	        #sFB_MCOConveyLinxAixController_110(iUDT_AixConfig          := #iqUDT_Configuration."110".MCO_M01,
	                                            iv_AixInputsModule    := #iUDT_MotorInput110,
	                                            ix_24vOk                := #ix_24vOk,
	                                            ix_SimulationModeActive := "DB_Memory".Simulation,
	                                            ii_MotorPositionId      := 1,
	                                            qUDT_HMIStatus          => #iqUDT_WorkstationStatus."110".MCO_M01,
	                                            iqv_AixOutputsModule  := #iqUDT_MotorOutput110,
	                                            iqUDT_ConveyorInterface := #sUDT_Interface_110,
	                                            iqUDT_MCOStatistics     := #iqUDT_WorkstationStatistics."110".MCO_M01);
	    END_REGION

	END_REGION

	REGION 120

	    REGION Displacement
	        #sFB_Displacement120(#sUDT_Interface_120);
	    END_REGION

	    REGION Tracking

	        #sFB_Tracking_120(iUDT_ConveyorCommonConfiguration := #iqUDT_Configuration."120".Conveyor.Common,
	                          iqa_TrackingData                 := #sa_TrackingArray_120,
	                          iqUDT_ConveyorInterface          := #sUDT_Interface_120,
	                          iqUDT_HandshakeUp                := #sUDT_Handshake_110,
	                          iqUDT_Handshake                  := #sUDT_Handshake_120);

	    END_REGION

	    REGION EoS

	        #sFB_PECUpdate_120(iUDT_PECUpdateConfiguration      := #iqUDT_Configuration."120".PEC_EoS,
	                           iUDT_ConveyorCommonConfiguration := #iqUDT_Configuration."120".Conveyor.Common,
	                           ix_PEC                           := #iUDT_MotorInput110.AllSensorPortInputs.RightSensor,
	                           ix_TeachingMode                  := FALSE,
	                           qUDT_Status                      => #iqUDT_WorkstationStatus."120".PEC_EoS,
	                           iqUDT_ConveyorInterface          := #sUDT_Interface_120,
	                           iqUDT_UnknownGINRange            := #iqUDT_UnknownGINRange,
	                           iqUDT_FifoHeader                 := #sUDT_FifoLostGINHeader,
	                           iqUDT_Statistics                 := #iqUDT_WorkstationStatistics."120".PEC_EoS,
	                           iqa_TrackingData                 := #sa_TrackingArray_120,
	                           iqa_FifoData                     := #sa_FifoLostGINData);

	    END_REGION

	    REGION Conveyor

	        #sFB_Conveyor_120(iUDT_ConveyorConfiguration := #iqUDT_Configuration."120".Conveyor,
	                          idi_PECEoSDistance         := #iqUDT_Configuration."120".PEC_EoS.Distance,
	                          idi_PECBoSDistance         := 0,
	                          ii_ExternalSpeed           := 0,
	                          ix_SafetyOk                := #ix_SafetyOk,
	                          ix_24vOk                   := #ix_24vOk,
	                          ix_400vOk                  := #ix_400vOk,
	                          ix_HardwareOk              := #iUDT_HardwareOk."110",
	                          ix_PECEoS                  := #iqUDT_WorkstationStatus."120".PEC_EoS.PEC,
	                          ix_PECBoS                  := TRUE,
	                          ix_ReverseDirection        := FALSE,
	                          ix_ExternalRequestDieBack  := #sx_Hold120 OR (#sUDT_Interface_130.ActualSpeed = 0 AND NOT #iqUDT_WorkstationStatus."120".PEC_EoS.PEC),
	                          ix_ExternalRequestHold     := FALSE,
	                          ix_ResetEnergySave         := FALSE,
	                          qUDT_HMIStatus             => #iqUDT_WorkstationStatus."120".Conveyor,
	                          qUDT_Status                => #iqUDT_WorkstationCommonStatus."120",
	                          iqUDT_EquipmentControl     := #iqUDT_EquipmentControl,
	                          iqUDT_ConveyorCommand      := #iqUDT_WorkstationCommands."120".Conveyor,
	                          iqUDT_ConveyorInterface    := #sUDT_Interface_120,
	                          iqUDT_HandShakeUp          := #sUDT_Handshake_110,
	                          iqUDT_HandShake            := #sUDT_Handshake_120,
	                          iqUDT_Statistics           := #iqUDT_WorkstationStatistics."120".Conveyor);

	    END_REGION

	    REGION MCO

	        #sFB_MCOConveyLinxAixController_120(iUDT_AixConfig          := #iqUDT_Configuration."120".MCO_M01,
	                                            iv_AixInputsModule    := #iUDT_MotorInput110,
	                                            ix_24vOk                := #ix_24vOk,
	                                            ix_SimulationModeActive := "DB_Memory".Simulation,
	                                            ii_MotorPositionId      := 2,
	                                            qUDT_HMIStatus          => #iqUDT_WorkstationStatus."120".MCO_M01,
	                                            iqv_AixOutputsModule  := #iqUDT_MotorOutput110,
	                                            iqUDT_ConveyorInterface := #sUDT_Interface_120,
	                                            iqUDT_MCOStatistics     := #iqUDT_WorkstationStatistics."120".MCO_M01);
	    END_REGION

	END_REGION

	REGION 130

	    REGION Displacement
	        #sFB_Displacement130(#sUDT_Interface_130);
	    END_REGION

	    REGION Tracking

	        #sFB_Tracking_130(iUDT_ConveyorCommonConfiguration := #iqUDT_Configuration."130".Conveyor.Common,
	                          iqa_TrackingData                 := #sa_TrackingArray_130,
	                          iqUDT_ConveyorInterface          := #sUDT_Interface_130,
	                          iqUDT_HandshakeUp                := #sUDT_Handshake_120,
	                          iqUDT_Handshake                  := #sUDT_Handshake_130);

	    END_REGION

	    REGION EoS

	        #sFB_PECUpdate_130(iUDT_PECUpdateConfiguration      := #iqUDT_Configuration."130".PEC_EoS,
	                           iUDT_ConveyorCommonConfiguration := #iqUDT_Configuration."130".Conveyor.Common,
	                           ix_PEC                           := #iUDT_MotorInput130.AllSensorPortInputs.LeftSensor,
	                           ix_TeachingMode                  := FALSE,
	                           qUDT_Status                      => #iqUDT_WorkstationStatus."130".PEC_EoS,
	                           iqUDT_ConveyorInterface          := #sUDT_Interface_130,
	                           iqUDT_UnknownGINRange            := #iqUDT_UnknownGINRange,
	                           iqUDT_FifoHeader                 := #sUDT_FifoLostGINHeader,
	                           iqUDT_Statistics                 := #iqUDT_WorkstationStatistics."130".PEC_EoS,
	                           iqa_TrackingData                 := #sa_TrackingArray_130,
	                           iqa_FifoData                     := #sa_FifoLostGINData);

	    END_REGION

	    REGION Conveyor

	        #sUDT_Handshake_130.RTR := #sUDT_Handshake_130.RTR AND NOT #sx_Hold130 OR #iqUDT_WorkstationStatus."130".PEC_EoS.PEC;

	        #sFB_Conveyor_130(iUDT_ConveyorConfiguration := #iqUDT_Configuration."130".Conveyor,
	                          idi_PECEoSDistance         := #iqUDT_Configuration."130".PEC_EoS.Distance,
	                          idi_PECBoSDistance         := 0,
	                          ii_ExternalSpeed           := 0,
	                          ix_SafetyOk                := #ix_SafetyOk,
	                          ix_24vOk                   := #ix_24vOk,
	                          ix_400vOk                  := #ix_400vOk,
	                          ix_HardwareOk              := #iUDT_HardwareOk."130",
	                          ix_PECEoS                  := #iqUDT_WorkstationStatus."130".PEC_EoS.PEC,
	                          ix_PECBoS                  := TRUE,
	                          ix_ReverseDirection        := FALSE,
	                          ix_ExternalRequestDieBack  := FALSE,
	                          ix_ExternalRequestHold     := #sx_Hold130,
	                          ix_ResetEnergySave         := FALSE,
	                          qUDT_HMIStatus             => #iqUDT_WorkstationStatus."130".Conveyor,
	                          qUDT_Status                => #iqUDT_WorkstationCommonStatus."130",
	                          iqUDT_EquipmentControl     := #iqUDT_EquipmentControl,
	                          iqUDT_ConveyorCommand      := #iqUDT_WorkstationCommands."130".Conveyor,
	                          iqUDT_ConveyorInterface    := #sUDT_Interface_130,
	                          iqUDT_HandShakeUp          := #sUDT_Handshake_120,
	                          iqUDT_HandShake            := #sUDT_Handshake_130,
	                          iqUDT_Statistics           := #iqUDT_WorkstationStatistics."130".Conveyor);


	    END_REGION

	    REGION MCO

	        #sFB_MCOConveyLinxAixController_130(iUDT_AixConfig          := #iqUDT_Configuration."130".MCO_M01,
	                                            iv_AixInputsModule    := #iUDT_MotorInput130,
	                                            ix_24vOk                := #ix_24vOk,
	                                            ix_SimulationModeActive := "DB_Memory".Simulation,
	                                            ii_MotorPositionId      := 1,
	                                            qUDT_HMIStatus          => #iqUDT_WorkstationStatus."130".MCO_M01,
	                                            iqv_AixOutputsModule  := #iqUDT_MotorOutput130,
	                                            iqUDT_ConveyorInterface := #sUDT_Interface_130,
	                                            iqUDT_MCOStatistics     := #iqUDT_WorkstationStatistics."130".MCO_M01);
	    END_REGION

	END_REGION

	REGION 140

	    REGION Displacement
	        #sFB_Displacement140(#sUDT_Interface_140);
	    END_REGION

	    REGION MCO

	        #sFB_MCOConveyLinxAixController_140(iUDT_AixConfig          := #iqUDT_Configuration."140".MCO_M01,
	                                            iv_AixInputsModule    := #iUDT_MotorInput140,
	                                            ii_PositionSetpoint     := #iqUDT_RATPositioning140.Lower.EndPosition,
	                                            ix_24vOk                := #ix_24vOk,
	                                            ix_SimulationModeActive := "DB_Memory".Simulation,
	                                            ii_MotorPositionId      := 1,
	                                            ix_StartPositioning     := #iqUDT_RATPositioning140.Lower.Start,
	                                            ix_ResetPosition        := #iqUDT_RATPositioning140.Lower.ResetPosition,
	                                            qUDT_HMIStatus          => #iqUDT_WorkstationStatus."140".MCO_M01,
	                                            qx_Positioned           => #iqUDT_RATPositioning140.Lower.Done,
	                                            iqv_AixOutputsModule  := #iqUDT_MotorOutput140,
	                                            iqUDT_ConveyorInterface := #sUDT_Interface_140,
	                                            iqUDT_MCOStatistics     := #iqUDT_WorkstationStatistics."140".MCO_M01);
	    END_REGION

	    REGION BladeStopEoS

	        IF (#iqUDT_Configuration.GlobalConfig.StationVariant = 2 OR #iqUDT_Configuration.GlobalConfig.StationVariant = 4 OR #iqUDT_Configuration.GlobalConfig.StationVariant = 6) THEN

	            #sFB_BladeStopEoS_140(iUDT_Configuration     := #iqUDT_Configuration."140".BladeStopEoS,
	                                  ix_IsOpened            := #ix_BladeStopIsUp140,
	                                  ix_IsClosed            := #ix_BladeStopIsDown140,
	                                  ix_AirPressureOk       := TRUE,
	                                  qx_Open                => #qx_BladeStopControl140,
	                                  qUDT_HMIStatus         => #iqUDT_WorkstationStatus."140".BladeStopEoS,
	                                  iqUDT_Statistics       := #iqUDT_WorkstationStatistics."140".BladeStopEoS,
	                                  iqUDT_EquipmentControl := #iqUDT_EquipmentControl,
	                                  iqUDT_HMICommand       := #iqUDT_WorkstationCommands."140".BladeStopEoS,
	                                  iqUDT_Interface        := #sUDT_Interface_140_BladeStopEoS);
	        END_IF;

	    END_REGION

	END_REGION

	REGION 141

	    REGION Displacement
	        #sFB_Displacement141(#sUDT_Interface_141);
	    END_REGION

	    REGION RAT

	        // #iqUDT_Configuration."141".RightAngledTransfer.BladeStop := #iqUDT_Configuration.GlobalConfig.StationVariant = 1
	        // OR #iqUDT_Configuration.GlobalConfig.StationVariant = 2
	        // OR #iqUDT_Configuration.GlobalConfig.StationVariant = 3
	        // OR #iqUDT_Configuration.GlobalConfig.StationVariant = 4;


	        IF #iqUDT_Configuration.GlobalConfig.StationVariant = 1 OR #iqUDT_Configuration.GlobalConfig.StationVariant = 3 OR #iqUDT_Configuration.GlobalConfig.StationVariant = 5 THEN
	            #sUDT_Handshake_141D := #sUDT_Handshake_241D;
	        ELSIF #iqUDT_Configuration.GlobalConfig.StationVariant = 2 OR #iqUDT_Configuration.GlobalConfig.StationVariant = 4 OR #iqUDT_Configuration.GlobalConfig.StationVariant = 6 THEN
	            #sUDT_Handshake_141C := #sUDT_Handshake_241C;
	        END_IF;

	        #sFB_RightAngledTransfer_141(iUDT_Configuration              := #iqUDT_Configuration."141".RightAngledTransfer,
	                                     iUDT_LowerConveyorConfiguration := #iqUDT_Configuration."140".Conveyor,
	                                     iUDT_UpperConveyorConfiguration := #iqUDT_Configuration."141".Conveyor,
	                                     iUDT_PECConfiguration           := #iqUDT_Configuration."140".PEC_EoS,
	                                     ii_DestinationA                 := #si_140DestinationA,
	                                     ii_DestinationB                 := #si_140DestinationB,
	                                     ii_DestinationC                 := #si_140DestinationC,
	                                     ii_DestinationD                 := #si_140DestinationD,
	                                     ix_HardwareOk                   := #iUDT_HardwareOk."140",
	                                     ix_400vOk                       := #ix_400vOk,
	                                     ix_24vOk                        := #ix_24vOk,
	                                     ix_SafetyOk                     := #ix_SafetyOk,
	                                     ix_AirPressureOk                := #ix_AirPressureOk,
	                                     ix_SectionIsDown                := #ix_SectionIsDown141,
	                                     ix_SectionIsUp                  := #ix_SectionIsUp141,
	                                     ix_ConveyorAAuto                := #iqUDT_WorkstationCommonStatus."130".AutoON,
	                                     ix_ConveyorBAuto                := #iqUDT_WorkstationCommonStatus."150".AutoON,
	                                     ix_ConveyorCAuto                := #iqUDT_WorkstationCommonStatus."241".AutoON AND (#iqUDT_Configuration.GlobalConfig.StationVariant = 2 OR #iqUDT_Configuration.GlobalConfig.StationVariant = 4 OR #iqUDT_Configuration.GlobalConfig.StationVariant = 6),
	                                     ix_ConveyorDAuto                := #iqUDT_WorkstationCommonStatus."241".AutoON AND (#iqUDT_Configuration.GlobalConfig.StationVariant = 1 OR #iqUDT_Configuration.GlobalConfig.StationVariant = 3 OR #iqUDT_Configuration.GlobalConfig.StationVariant = 5),
	                                     ix_PEC                          := #iUDT_MotorInput140.AllSensorPortInputs.LeftSensor,
	                                     ix_ExternalReceiveRequestA      := NOT #iqUDT_WorkstationStatus."130".PEC_EoS.PEC AND #sx_Enable1X0In,
	                                     ix_ExternalReceiveRequestB      := false,
	                                     ix_ExternalReceiveRequestC      := #sFB_RightAngledTransfer_241.qx_ExternalSendRequestC AND (#iqUDT_Configuration.GlobalConfig.StationVariant = 2 OR #iqUDT_Configuration.GlobalConfig.StationVariant = 4 OR #iqUDT_Configuration.GlobalConfig.StationVariant = 6),
	                                     ix_ExternalReceiveRequestD      := #sFB_RightAngledTransfer_241.qx_ExternalSendRequestD AND (#iqUDT_Configuration.GlobalConfig.StationVariant = 1 OR #iqUDT_Configuration.GlobalConfig.StationVariant = 3 OR #iqUDT_Configuration.GlobalConfig.StationVariant = 5),
	                                     ix_PECInfeedA                   := #iqUDT_WorkstationStatus."130".PEC_EoS.PEC,
	                                     ix_PECInfeedC                   := #iqUDT_WorkstationStatus."240".PEC_EoS.PEC AND (#iqUDT_Configuration.GlobalConfig.StationVariant = 2 OR #iqUDT_Configuration.GlobalConfig.StationVariant = 4 OR #iqUDT_Configuration.GlobalConfig.StationVariant = 6),
	                                     ix_PECInfeedD                   := #iqUDT_WorkstationStatus."240".PEC_EoS.PEC AND (#iqUDT_Configuration.GlobalConfig.StationVariant = 1 OR #iqUDT_Configuration.GlobalConfig.StationVariant = 3 OR #iqUDT_Configuration.GlobalConfig.StationVariant = 5),
	                                     qUDT_HMIRATStatus               => #iqUDT_WorkstationStatus."141".RightAngledTransfer,
	                                     qUDT_HMIConveyorStatus          => #iqUDT_WorkstationStatus."140".Conveyor,
	                                     qUDT_HMIPECStatus               => #iqUDT_WorkstationStatus."140".PEC_EoS,
	                                     qUDT_RATStatus                  => #iqUDT_WorkstationCommonStatus."141",
	                                     qUDT_ConveyorStatus             => #iqUDT_WorkstationCommonStatus."140",
	                                     qx_PopupControl                 => #qx_PopupControl141,
	                                     iqUDT_EquipmentControl          := #iqUDT_EquipmentControl,
	                                     iqUDT_RATCommand                := #iqUDT_WorkstationCommands."141".RightAngledTransfer,
	                                     iqUDT_ConveyorCommand           := #iqUDT_WorkstationCommands."140".Conveyor,
	                                     iqUDT_RATStatistics             := #iqUDT_WorkstationStatistics."141".RightAngledTransfer,
	                                     iqUDT_ConveyorStatistics        := #iqUDT_WorkstationStatistics."140".Conveyor,
	                                     iqUDT_PECStatistics             := #iqUDT_WorkstationStatistics."140".PEC_EoS,
	                                     iqUDT_HandShakeConveyorA        := #sUDT_Handshake_130,
	                                     iqUDT_HandShakeConveyorB        := #sUDT_Handshake_140,
	                                     iqUDT_HandShakeConveyorC        := #sUDT_Handshake_141C,
	                                     iqUDT_HandShakeConveyorD        := #sUDT_Handshake_141D,
	                                     iqUDT_LowerConveyorInterface    := #sUDT_Interface_140,
	                                     iqUDT_UpperConveyorInterface    := #sUDT_Interface_141,
	                                     iqUDT_RATPositioning            := #iqUDT_RATPositioning140,
	                                     iqUDT_BladeStopEoSInterface     := #sUDT_Interface_140_BladeStopEoS,
	                                     iqUDT_BladeStopBoSInterface     := #tUDT_DummyBladeStop);

	    END_REGION

	    IF #iqUDT_Configuration.GlobalConfig.StationVariant = 1 OR #iqUDT_Configuration.GlobalConfig.StationVariant = 3 OR #iqUDT_Configuration.GlobalConfig.StationVariant = 5 THEN

	        #sUDT_Handshake_241D := #sUDT_Handshake_141D;
	    ELSIF #iqUDT_Configuration.GlobalConfig.StationVariant = 2 OR #iqUDT_Configuration.GlobalConfig.StationVariant = 4 OR #iqUDT_Configuration.GlobalConfig.StationVariant = 6 THEN
	        #sUDT_Handshake_241C := #sUDT_Handshake_141C;

	    END_IF;

	    REGION MCO

	        #sFB_MCOConveyLinxAixController_141(iUDT_AixConfig          := #iqUDT_Configuration."141".MCO_M01,
	                                            iv_AixInputsModule    := #iUDT_MotorInput140,
	                                            ii_PositionSetpoint     := #iqUDT_RATPositioning140.Upper.EndPosition,
	                                            ix_24vOk                := #ix_24vOk,
	                                            ix_SimulationModeActive := "DB_Memory".Simulation,
	                                            ii_MotorPositionId      := 2,
	                                            ix_StartPositioning     := #iqUDT_RATPositioning140.Upper.Start,
	                                            ix_ResetPosition        := #iqUDT_RATPositioning140.Upper.ResetPosition,
	                                            qUDT_HMIStatus          => #iqUDT_WorkstationStatus."141".MCO_M01,
	                                            qx_Positioned           => #iqUDT_RATPositioning140.Upper.Done,
	                                            iqv_AixOutputsModule  := #iqUDT_MotorOutput140,
	                                            iqUDT_ConveyorInterface := #sUDT_Interface_141,
	                                            iqUDT_MCOStatistics     := #iqUDT_WorkstationStatistics."141".MCO_M01);
	    END_REGION

	END_REGION

	IF #iqUDT_Configuration.GlobalConfig.StationVariant = 1 OR #iqUDT_Configuration.GlobalConfig.StationVariant = 2 OR #iqUDT_Configuration.GlobalConfig.StationVariant = 3 OR #iqUDT_Configuration.GlobalConfig.StationVariant = 4 THEN

	    REGION 150

	        REGION Displacement
	            #sFB_Displacement150(#sUDT_Interface_150);
	        END_REGION

	        REGION Tracking

	            #sFB_Tracking_150(iUDT_ConveyorCommonConfiguration := #iqUDT_Configuration."150".Conveyor.Common,
	                              iqa_TrackingData                 := #sa_TrackingArray_150,
	                              iqUDT_ConveyorInterface          := #sUDT_Interface_150,
	                              iqUDT_HandshakeUp                := #sUDT_Handshake_140,
	                              iqUDT_Handshake                  := #sUDT_Handshake_150);

	        END_REGION

	        REGION EoS

	            #sFB_PECUpdate_150(iUDT_PECUpdateConfiguration      := #iqUDT_Configuration."150".PEC_EoS,
	                               iUDT_ConveyorCommonConfiguration := #iqUDT_Configuration."150".Conveyor.Common,
	                               ix_PEC                           := NOT #iUDT_MotorInput150.AllSensorPortInputs.LeftSensor,
	                               ix_TeachingMode                  := FALSE,
	                               qUDT_Status                      => #iqUDT_WorkstationStatus."150".PEC_EoS,
	                               iqUDT_ConveyorInterface          := #sUDT_Interface_150,
	                               iqUDT_UnknownGINRange            := #iqUDT_UnknownGINRange,
	                               iqUDT_FifoHeader                 := #sUDT_FifoLostGINHeader,
	                               iqUDT_Statistics                 := #iqUDT_WorkstationStatistics."150".PEC_EoS,
	                               iqa_TrackingData                 := #sa_TrackingArray_150,
	                               iqa_FifoData                     := #sa_FifoLostGINData);




	        END_REGION

	        REGION Conveyor

	            //  #sUDT_Handshake_150.RTR := true;
	            // #tx_Enable := (#iqUDT_WorkstationStatus."160".PEC_EoS.PEC AND #sUDT_Interface_160.ActualSpeed <> 0)
	            // OR (#iqUDT_WorkstationStatus."150".PEC_EoS.PEC);
	            #sUDT_Handshake_150.RTR := (#iqUDT_WorkstationStatus."160".PEC_EoS.PEC AND #sUDT_Interface_160.ActualSpeed <> 0)
	            OR (#iqUDT_WorkstationStatus."150".PEC_EoS.PEC);
	            #sFB_Conveyor_150(iUDT_ConveyorConfiguration := #iqUDT_Configuration."150".Conveyor,
	                              idi_PECEoSDistance         := #iqUDT_Configuration."150".PEC_EoS.Distance,
	                              idi_PECBoSDistance         := 0,
	                              ii_ExternalSpeed           := 0,
	                              ix_SafetyOk                := #ix_SafetyOk,
	                              ix_24vOk                   := #ix_24vOk,
	                              ix_400vOk                  := #ix_400vOk,
	                              ix_HardwareOk              := #iUDT_HardwareOk."150",
	                              ix_PECEoS                  := #iqUDT_WorkstationStatus."150".PEC_EoS.PEC,
	                              ix_PECBoS                  := TRUE,
	                              ix_ReverseDirection        := FALSE,
	                              ix_ExternalRequestDieBack  := FALSE,
	                              ix_ExternalRequestHold     := #sx_ReleaseBinHold1X0,//sx_Hold150,//NOT #tx_Enable,
	                              ix_ResetEnergySave         := FALSE,
	                              qUDT_HMIStatus             => #iqUDT_WorkstationStatus."150".Conveyor,
	                              qUDT_Status                => #iqUDT_WorkstationCommonStatus."150",
	                              iqUDT_EquipmentControl     := #iqUDT_EquipmentControl,
	                              iqUDT_ConveyorCommand      := #iqUDT_WorkstationCommands."150".Conveyor,
	                              iqUDT_ConveyorInterface    := #sUDT_Interface_150,
	                              iqUDT_HandShakeUp          := #sUDT_Handshake_140,
	                              iqUDT_HandShake            := #sUDT_Handshake_150,
	                              iqUDT_Statistics           := #iqUDT_WorkstationStatistics."150".Conveyor);

	        END_REGION

	        REGION MCO

	            #sFB_MCOConveyLinxAixController_150(iUDT_AixConfig          := #iqUDT_Configuration."150".MCO_M01,
	                                                iv_AixInputsModule    := #iUDT_MotorInput150,
	                                                ix_24vOk                := #ix_24vOk,
	                                                ix_SimulationModeActive := "DB_Memory".Simulation,
	                                                ii_MotorPositionId      := 1,
	                                                qUDT_HMIStatus          => #iqUDT_WorkstationStatus."150".MCO_M01,
	                                                iqv_AixOutputsModule  := #iqUDT_MotorOutput150,
	                                                iqUDT_ConveyorInterface := #sUDT_Interface_150,
	                                                iqUDT_MCOStatistics     := #iqUDT_WorkstationStatistics."150".MCO_M01);
	        END_REGION

	    END_REGION

	    REGION 160

	        REGION Displacement
	            #sFB_Displacement160(#sUDT_Interface_160);
	        END_REGION

	        REGION Tracking

	            #sFB_Tracking_160(iUDT_ConveyorCommonConfiguration := #iqUDT_Configuration."160".Conveyor.Common,
	                              iqa_TrackingData                 := #sa_TrackingArray_160,
	                              iqUDT_ConveyorInterface          := #sUDT_Interface_160,
	                              iqUDT_HandshakeUp                := #sUDT_Handshake_150,
	                              iqUDT_Handshake                  := #sUDT_Handshake_160);

	        END_REGION

	        REGION EoS

	            #sFB_PECUpdate_160(iUDT_PECUpdateConfiguration      := #iqUDT_Configuration."160".PEC_EoS,
	                               iUDT_ConveyorCommonConfiguration := #iqUDT_Configuration."160".Conveyor.Common,
	                               ix_PEC                           := NOT #iUDT_MotorInput150.AllSensorPortInputs.RightSensor,
	                               ix_TeachingMode                  := FALSE,
	                               qUDT_Status                      => #iqUDT_WorkstationStatus."160".PEC_EoS,
	                               iqUDT_ConveyorInterface          := #sUDT_Interface_160,
	                               iqUDT_UnknownGINRange            := #iqUDT_UnknownGINRange,
	                               iqUDT_FifoHeader                 := #sUDT_FifoLostGINHeader,
	                               iqUDT_Statistics                 := #iqUDT_WorkstationStatistics."160".PEC_EoS,
	                               iqa_TrackingData                 := #sa_TrackingArray_160,
	                               iqa_FifoData                     := #sa_FifoLostGINData);




	        END_REGION

	        REGION Conveyor

	            // #sUDT_Handshake_160.RTR := true;
	            // #tx_Enable := (#iqUDT_WorkstationStatus."170".PEC_EoS.PEC AND #sUDT_Interface_170.ActualSpeed <> 0)
	            //  OR (#iqUDT_WorkstationStatus."160".PEC_EoS.PEC);
	            #sUDT_Handshake_160.RTR := (#iqUDT_WorkstationStatus."170".PEC_EoS.PEC AND #sUDT_Interface_170.ActualSpeed <> 0)
	            OR (#iqUDT_WorkstationStatus."160".PEC_EoS.PEC);


	            #sFB_Conveyor_160(iUDT_ConveyorConfiguration := #iqUDT_Configuration."160".Conveyor,
	                              idi_PECEoSDistance         := #iqUDT_Configuration."160".PEC_EoS.Distance,
	                              idi_PECBoSDistance         := 0,
	                              ii_ExternalSpeed           := 0,
	                              ix_SafetyOk                := #ix_SafetyOk,
	                              ix_24vOk                   := #ix_24vOk,
	                              ix_400vOk                  := #ix_400vOk,
	                              ix_HardwareOk              := #iUDT_HardwareOk."150",
	                              ix_PECEoS                  := #iqUDT_WorkstationStatus."160".PEC_EoS.PEC,
	                              ix_PECBoS                  := TRUE,
	                              ix_ReverseDirection        := FALSE,
	                              ix_ExternalRequestDieBack  := FALSE,
	                              ix_ExternalRequestHold     := #sx_Hold160,//NOT #tx_Enable,//NOT #iqUDT_WorkstationStatus."160"."132".PEC_EoS.PEC AND NOT #iqUDT_WorkstationStatus."135"."136".PEC_EoS.PEC AND NOT (#sUDT_Interface_170.ActualSpeed <> 0),
	                              ix_ResetEnergySave         := FALSE,
	                              qUDT_HMIStatus             => #iqUDT_WorkstationStatus."160".Conveyor,
	                              qUDT_Status                => #iqUDT_WorkstationCommonStatus."160",
	                              iqUDT_EquipmentControl     := #iqUDT_EquipmentControl,
	                              iqUDT_ConveyorCommand      := #iqUDT_WorkstationCommands."160".Conveyor,
	                              iqUDT_ConveyorInterface    := #sUDT_Interface_160,
	                              iqUDT_HandShakeUp          := #sUDT_Handshake_150,
	                              iqUDT_HandShake            := #sUDT_Handshake_160,
	                              iqUDT_Statistics           := #iqUDT_WorkstationStatistics."160".Conveyor);

	        END_REGION

	        REGION MCO

	            #sFB_MCOConveyLinxAixController_160(iUDT_AixConfig          := #iqUDT_Configuration."160".MCO_M01,
	                                                iv_AixInputsModule    := #iUDT_MotorInput150,
	                                                ix_24vOk                := #ix_24vOk,
	                                                ix_SimulationModeActive := "DB_Memory".Simulation,
	                                                ii_MotorPositionId      := 2,
	                                                qUDT_HMIStatus          => #iqUDT_WorkstationStatus."160".MCO_M01,
	                                                iqv_AixOutputsModule  := #iqUDT_MotorOutput150,
	                                                iqUDT_ConveyorInterface := #sUDT_Interface_160,
	                                                iqUDT_MCOStatistics     := #iqUDT_WorkstationStatistics."160".MCO_M01);
	        END_REGION

	    END_REGION

	    REGION 170

	        REGION Displacement
	            #sFB_Displacement170(#sUDT_Interface_170);
	        END_REGION

	        REGION Tracking

	            #sFB_Tracking_170(iUDT_ConveyorCommonConfiguration := #iqUDT_Configuration."170".Conveyor.Common,
	                              iqa_TrackingData                 := #sa_TrackingArray_170,
	                              iqUDT_ConveyorInterface          := #sUDT_Interface_170,
	                              iqUDT_HandshakeUp                := #sUDT_Handshake_160,
	                              iqUDT_Handshake                  := #sUDT_Handshake_170);

	        END_REGION

	        REGION EoS

	            #sFB_PECUpdate_170(iUDT_PECUpdateConfiguration      := #iqUDT_Configuration."170".PEC_EoS,
	                               iUDT_ConveyorCommonConfiguration := #iqUDT_Configuration."170".Conveyor.Common,
	                               ix_PEC                           := NOT #iUDT_MotorInput170.AllSensorPortInputs.LeftSensor,
	                               ix_TeachingMode                  := FALSE,
	                               qUDT_Status                      => #iqUDT_WorkstationStatus."170".PEC_EoS,
	                               iqUDT_ConveyorInterface          := #sUDT_Interface_170,
	                               iqUDT_UnknownGINRange            := #iqUDT_UnknownGINRange,
	                               iqUDT_FifoHeader                 := #sUDT_FifoLostGINHeader,
	                               iqUDT_Statistics                 := #iqUDT_WorkstationStatistics."170".PEC_EoS,
	                               iqa_TrackingData                 := #sa_TrackingArray_170,
	                               iqa_FifoData                     := #sa_FifoLostGINData);

	        END_REGION

	        REGION Conveyor



	            #sUDT_Handshake_170.RTR := #iqUDT_WorkstationStatus."170".PEC_EoS.PEC;

	            #sFB_Conveyor_170(iUDT_ConveyorConfiguration := #iqUDT_Configuration."170".Conveyor,
	                              idi_PECEoSDistance         := #iqUDT_Configuration."170".PEC_EoS.Distance,
	                              idi_PECBoSDistance         := 0,
	                              ii_ExternalSpeed           := 0,
	                              ix_SafetyOk                := #ix_SafetyOk,
	                              ix_24vOk                   := #ix_24vOk,
	                              ix_400vOk                  := #ix_400vOk,
	                              ix_HardwareOk              := #iUDT_HardwareOk."170",
	                              ix_PECEoS                  := #iqUDT_WorkstationStatus."170".PEC_EoS.PEC,
	                              ix_PECBoS                  := TRUE,
	                              ix_ReverseDirection        := FALSE,
	                              ix_ExternalRequestDieBack  := FALSE,
	                              ix_ExternalRequestHold     := #sx_Hold170,
	                              ix_ResetEnergySave         := FALSE,
	                              qUDT_HMIStatus             => #iqUDT_WorkstationStatus."170".Conveyor,
	                              qUDT_Status                => #iqUDT_WorkstationCommonStatus."170",
	                              iqUDT_EquipmentControl     := #iqUDT_EquipmentControl,
	                              iqUDT_ConveyorCommand      := #iqUDT_WorkstationCommands."170".Conveyor,
	                              iqUDT_ConveyorInterface    := #sUDT_Interface_170,
	                              iqUDT_HandShakeUp          := #sUDT_Handshake_160,
	                              iqUDT_HandShake            := #sUDT_Handshake_170,
	                              iqUDT_Statistics           := #iqUDT_WorkstationStatistics."170".Conveyor);

	        END_REGION

	        REGION MCO

	            #sFB_MCOConveyLinxAixController_170(iUDT_AixConfig          := #iqUDT_Configuration."170".MCO_M01,
	                                                iv_AixInputsModule    := #iUDT_MotorInput170,
	                                                ix_24vOk                := #ix_24vOk,
	                                                ix_SimulationModeActive := "DB_Memory".Simulation,
	                                                ii_MotorPositionId      := 1,
	                                                qUDT_HMIStatus          => #iqUDT_WorkstationStatus."170".MCO_M01,
	                                                iqv_AixOutputsModule  := #iqUDT_MotorOutput170,
	                                                iqUDT_ConveyorInterface := #sUDT_Interface_170,
	                                                iqUDT_MCOStatistics     := #iqUDT_WorkstationStatistics."170".MCO_M01);
	        END_REGION
	    END_REGION

	    REGION 180

	        REGION Displacement
	            #sFB_Displacement180(#sUDT_Interface_180);
	        END_REGION
	        (*
	        REGION EoS
	            #sFB_PEC_180(ix_PEC                  := #iUDT_MotorInput170.AllSensorPortInputs.RightSensor,
	                         iUDT_PECConfiguration   := #iqUDT_Configuration."180".PEC_EoS,
	                         qUDT_HMIStatus          => #iqUDT_WorkstationStatus."180".PEC_EoS,
	                         iqUDT_ConveyorInterface := #sUDT_Interface_180,
	                         iqUDT_PECStatistics     := #iqUDT_WorkstationStatistics."180".PEC_EoS);
	        END_REGION
	        *)
	        REGION Conveyor

	            #sUDT_Handshake_180.RTR := TRUE;

	            #sFB_Conveyor_180(iUDT_ConveyorConfiguration := #iqUDT_Configuration."180".Conveyor,
	                              idi_PECEoSDistance         := 0,
	                              idi_PECBoSDistance         := 0,
	                              ii_ExternalSpeed           := 0,
	                              ix_SafetyOk                := #ix_SafetyOk,
	                              ix_24vOk                   := #ix_24vOk,
	                              ix_400vOk                  := #ix_400vOk,
	                              ix_HardwareOk              := #iUDT_HardwareOk."170",
	                              ix_PECEoS                  := TRUE,
	                              ix_PECBoS                  := TRUE,
	                              ix_ReverseDirection        := FALSE,
	                              ix_ExternalRequestDieBack  := FALSE,
	                              ix_ExternalRequestHold     := #sx_Hold180,
	                              ix_ResetEnergySave         := NOT #sx_Hold180,
	                              qUDT_HMIStatus             => #iqUDT_WorkstationStatus."180".Conveyor,
	                              qUDT_Status                => #iqUDT_WorkstationCommonStatus."180",
	                              iqUDT_EquipmentControl     := #iqUDT_EquipmentControl,
	                              iqUDT_ConveyorCommand      := #iqUDT_WorkstationCommands."180".Conveyor,
	                              iqUDT_ConveyorInterface    := #sUDT_Interface_180,
	                              iqUDT_HandShakeUp          := #sUDT_HandshakeUp_180,
	                              iqUDT_HandShake            := #sUDT_Handshake_180,
	                              iqUDT_Statistics           := #iqUDT_WorkstationStatistics."180".Conveyor);

	        END_REGION

	        REGION MCO

	            #sFB_MCOConveyLinxAixController_180(iUDT_AixConfig          := #iqUDT_Configuration."180".MCO_M01,
	                                                iv_AixInputsModule    := #iUDT_MotorInput170,
	                                                ix_24vOk                := #ix_24vOk,
	                                                ix_SimulationModeActive := "DB_Memory".Simulation,
	                                                ii_MotorPositionId      := 2,
	                                                qUDT_HMIStatus          => #iqUDT_WorkstationStatus."180".MCO_M01,
	                                                iqv_AixOutputsModule  := #iqUDT_MotorOutput170,
	                                                iqUDT_ConveyorInterface := #sUDT_Interface_180,
	                                                iqUDT_MCOStatistics     := #iqUDT_WorkstationStatistics."180".MCO_M01);
	        END_REGION

	    END_REGION
	END_IF;
	REGION 210

	    REGION Displacement
	        #sFB_Displacement210(#sUDT_Interface_210);
	    END_REGION

	    REGION EoS


	        #sFB_PEC_210(ix_PEC                  := NOT #iUDT_MotorInput210.AllSensorPortInputs.LeftSensor,
	                     iUDT_PECConfiguration   := #iqUDT_Configuration."210".PEC_EoS,
	                     qUDT_HMIStatus          => #iqUDT_WorkstationStatus."210".PEC_EoS,
	                     iqUDT_ConveyorInterface := #sUDT_Interface_210,
	                     iqUDT_PECStatistics     := #iqUDT_WorkstationStatistics."210".PEC_EoS);

	    END_REGION

	    REGION Conveyor

	        #sFB_Conveyor_210(iUDT_ConveyorConfiguration := #iqUDT_Configuration."210".Conveyor,
	                          idi_PECEoSDistance         := #iqUDT_Configuration."210".PEC_EoS.Distance,
	                          idi_PECBoSDistance         := 0,
	                          ii_ExternalSpeed           := 0,
	                          ix_SafetyOk                := #ix_SafetyOk,
	                          ix_24vOk                   := #ix_24vOk,
	                          ix_400vOk                  := #ix_400vOk,
	                          ix_HardwareOk              := #iUDT_HardwareOk."210",
	                          ix_PECEoS                  := #iqUDT_WorkstationStatus."210".PEC_EoS.PEC,
	                          ix_PECBoS                  := TRUE,
	                          ix_ReverseDirection        := FALSE,
	                          ix_ExternalRequestDieBack  := FALSE,
	                          ix_ExternalRequestHold     := #sx_ReleaseBinHold0X0 OR #sx_ReleaseBinHold1X0 OR NOT #sUDT_Handshake_210.RTR,
	                          ix_ResetEnergySave         := #sx_ReleaseBinHold0X0 OR #sx_ReleaseBinHold1X0,
	                          qUDT_HMIStatus             => #iqUDT_WorkstationStatus."210".Conveyor,
	                          qUDT_Status                => #iqUDT_WorkstationCommonStatus."210",
	                          iqUDT_EquipmentControl     := #iqUDT_EquipmentControl,
	                          iqUDT_ConveyorCommand      := #iqUDT_WorkstationCommands."210".Conveyor,
	                          iqUDT_ConveyorInterface    := #sUDT_Interface_210,
	                          iqUDT_HandShakeUp          := #sUDT_HandshakeUp_210,
	                          iqUDT_HandShake            := #sUDT_Handshake_210,
	                          iqUDT_Statistics           := #iqUDT_WorkstationStatistics."210".Conveyor);

	    END_REGION

	    REGION MCO

	        #sFB_MCOConveyLinxAixController_210(iUDT_AixConfig          := #iqUDT_Configuration."210".MCO_M01,
	                                            iv_AixInputsModule    := #iUDT_MotorInput210,
	                                            ix_24vOk                := #ix_24vOk,
	                                            ix_SimulationModeActive := "DB_Memory".Simulation,
	                                            ii_MotorPositionId      := 1,
	                                            qUDT_HMIStatus          => #iqUDT_WorkstationStatus."210".MCO_M01,
	                                            iqv_AixOutputsModule  := #iqUDT_MotorOutput210,
	                                            iqUDT_ConveyorInterface := #sUDT_Interface_210,
	                                            iqUDT_MCOStatistics     := #iqUDT_WorkstationStatistics."210".MCO_M01);
	    END_REGION

	END_REGION

	REGION 220

	    REGION Displacement
	        #sFB_Displacement220(#sUDT_Interface_220);
	    END_REGION



	    REGION EoS



	        #sFB_PEC_220(ix_PEC                  := NOT #iUDT_MotorInput210.AllSensorPortInputs.RightSensor,
	                     iUDT_PECConfiguration   := #iqUDT_Configuration."220".PEC_EoS,
	                     qUDT_HMIStatus          => #iqUDT_WorkstationStatus."220".PEC_EoS,
	                     iqUDT_ConveyorInterface := #sUDT_Interface_220,
	                     iqUDT_PECStatistics     := #iqUDT_WorkstationStatistics."220".PEC_EoS);


	    END_REGION

	    REGION Conveyor

	        #sFB_Conveyor_220(iUDT_ConveyorConfiguration := #iqUDT_Configuration."220".Conveyor,
	                          idi_PECEoSDistance         := #iqUDT_Configuration."220".PEC_EoS.Distance,
	                          idi_PECBoSDistance         := 0,
	                          ii_ExternalSpeed           := 0,
	                          ix_SafetyOk                := #ix_SafetyOk,
	                          ix_24vOk                   := #ix_24vOk,
	                          ix_400vOk                  := #ix_400vOk,
	                          ix_HardwareOk              := #iUDT_HardwareOk."210",
	                          ix_PECEoS                  := #iqUDT_WorkstationStatus."220".PEC_EoS.PEC,
	                          ix_PECBoS                  := TRUE,
	                          ix_ReverseDirection        := FALSE,
	                          ix_ExternalRequestDieBack  := FALSE,
	                          ix_ExternalRequestHold     := #sx_Hold220 OR #sx_ReleaseBinHold0X0 OR #sx_ReleaseBinHold1X0,
	                          ix_ResetEnergySave         := #sx_ReleaseBinHold0X0 OR #sx_ReleaseBinHold1X0,
	                          qUDT_HMIStatus             => #iqUDT_WorkstationStatus."220".Conveyor,
	                          qUDT_Status                => #iqUDT_WorkstationCommonStatus."220",
	                          iqUDT_EquipmentControl     := #iqUDT_EquipmentControl,
	                          iqUDT_ConveyorCommand      := #iqUDT_WorkstationCommands."220".Conveyor,
	                          iqUDT_ConveyorInterface    := #sUDT_Interface_220,
	                          iqUDT_HandShakeUp          := #sUDT_Handshake_210,
	                          iqUDT_HandShake            := #sUDT_Handshake_220,
	                          iqUDT_Statistics           := #iqUDT_WorkstationStatistics."220".Conveyor);

	    END_REGION

	    REGION MCO

	        #sFB_MCOConveyLinxAixController_220(iUDT_AixConfig          := #iqUDT_Configuration."220".MCO_M01,
	                                            iv_AixInputsModule    := #iUDT_MotorInput210,
	                                            ix_24vOk                := #ix_24vOk,
	                                            ix_SimulationModeActive := "DB_Memory".Simulation,
	                                            ii_MotorPositionId      := 2,
	                                            qUDT_HMIStatus          => #iqUDT_WorkstationStatus."220".MCO_M01,
	                                            iqv_AixOutputsModule  := #iqUDT_MotorOutput210,
	                                            iqUDT_ConveyorInterface := #sUDT_Interface_220,
	                                            iqUDT_MCOStatistics     := #iqUDT_WorkstationStatistics."220".MCO_M01);
	    END_REGION


	END_REGION

	REGION 230

	    REGION Displacement
	        #sFB_Displacement230(#sUDT_Interface_230);
	    END_REGION



	    REGION EoS




	        #sFB_PEC_230(ix_PEC                  := NOT #iUDT_MotorInput230.AllSensorPortInputs.LeftSensor,
	                     iUDT_PECConfiguration   := #iqUDT_Configuration."230".PEC_EoS,
	                     qUDT_HMIStatus          => #iqUDT_WorkstationStatus."230".PEC_EoS,
	                     iqUDT_ConveyorInterface := #sUDT_Interface_230,
	                     iqUDT_PECStatistics     := #iqUDT_WorkstationStatistics."230".PEC_EoS);




	    END_REGION

	    REGION Conveyor
	        #sUDT_Handshake_230.RTR := #sUDT_Handshake_230.RTR OR #iqUDT_WorkstationStatus."230".PEC_EoS.PEC;
	        #sFB_Conveyor_230(iUDT_ConveyorConfiguration := #iqUDT_Configuration."230".Conveyor,
	                          idi_PECEoSDistance         := #iqUDT_Configuration."230".PEC_EoS.Distance,
	                          idi_PECBoSDistance         := 0,
	                          ii_ExternalSpeed           := 0,
	                          ix_SafetyOk                := #ix_SafetyOk,
	                          ix_24vOk                   := #ix_24vOk,
	                          ix_400vOk                  := #ix_400vOk,
	                          ix_HardwareOk              := #iUDT_HardwareOk."230",
	                          ix_PECEoS                  := #iqUDT_WorkstationStatus."230".PEC_EoS.PEC,
	                          ix_PECBoS                  := TRUE,
	                          ix_ReverseDirection        := FALSE,
	                          ix_ExternalRequestDieBack  := FALSE,
	                          ix_ExternalRequestHold     := #sx_Hold230 OR #sx_ReleaseBinHold0X0 OR #sx_ReleaseBinHold1X0,
	                          ix_ResetEnergySave         := #sx_ReleaseBinHold0X0 OR #sx_ReleaseBinHold1X0,
	                          qUDT_HMIStatus             => #iqUDT_WorkstationStatus."230".Conveyor,
	                          qUDT_Status                => #iqUDT_WorkstationCommonStatus."230",
	                          iqUDT_EquipmentControl     := #iqUDT_EquipmentControl,
	                          iqUDT_ConveyorCommand      := #iqUDT_WorkstationCommands."230".Conveyor,
	                          iqUDT_ConveyorInterface    := #sUDT_Interface_230,
	                          iqUDT_HandShakeUp          := #sUDT_Handshake_220,
	                          iqUDT_HandShake            := #sUDT_Handshake_230,
	                          iqUDT_Statistics           := #iqUDT_WorkstationStatistics."230".Conveyor);

	    END_REGION

	    REGION MCO

	        #sFB_MCOConveyLinxAixController_230(iUDT_AixConfig          := #iqUDT_Configuration."230".MCO_M01,
	                                            iv_AixInputsModule    := #iUDT_MotorInput230,
	                                            ix_24vOk                := #ix_24vOk,
	                                            ix_SimulationModeActive := "DB_Memory".Simulation,
	                                            ii_MotorPositionId      := 1,
	                                            qUDT_HMIStatus          => #iqUDT_WorkstationStatus."230".MCO_M01,
	                                            iqv_AixOutputsModule  := #iqUDT_MotorOutput230,
	                                            iqUDT_ConveyorInterface := #sUDT_Interface_230,
	                                            iqUDT_MCOStatistics     := #iqUDT_WorkstationStatistics."230".MCO_M01);
	    END_REGION

	END_REGION

	REGION 240

	    REGION Displacement
	        #sFB_Displacement240(#sUDT_Interface_240);
	    END_REGION

	    REGION MCO

	        #sFB_MCOConveyLinxAixController_240(iUDT_AixConfig          := #iqUDT_Configuration."240".MCO_M01,
	                                            iv_AixInputsModule    := #iUDT_MotorInput240,
	                                            ii_PositionSetpoint     := #iqUDT_RATPositioning240.Lower.EndPosition,
	                                            ix_24vOk                := #ix_24vOk,
	                                            ix_SimulationModeActive := "DB_Memory".Simulation,
	                                            ii_MotorPositionId      := 1,
	                                            ix_StartPositioning     := #iqUDT_RATPositioning240.Lower.Start,
	                                            ix_ResetPosition        := #iqUDT_RATPositioning240.Lower.ResetPosition,
	                                            qUDT_HMIStatus          => #iqUDT_WorkstationStatus."240".MCO_M01,
	                                            qx_Positioned           => #iqUDT_RATPositioning240.Lower.Done,
	                                            iqv_AixOutputsModule  := #iqUDT_MotorOutput240,
	                                            iqUDT_ConveyorInterface := #sUDT_Interface_240,
	                                            iqUDT_MCOStatistics     := #iqUDT_WorkstationStatistics."240".MCO_M01);
	    END_REGION

	END_REGION

	REGION 241

	    REGION Displacement
	        #sFB_Displacement241(#sUDT_Interface_241);
	    END_REGION

	    REGION RAT

	        IF #iqUDT_Configuration.GlobalConfig.StationVariant = 1 OR #iqUDT_Configuration.GlobalConfig.StationVariant = 3 OR #iqUDT_Configuration.GlobalConfig.StationVariant = 5 THEN
	            #sUDT_Handshake_241C := #sUDT_Handshake_041C;
	            #sUDT_Handshake_241D := #sUDT_Handshake_141D;
	        ELSIF #iqUDT_Configuration.GlobalConfig.StationVariant = 2 OR #iqUDT_Configuration.GlobalConfig.StationVariant = 4 OR #iqUDT_Configuration.GlobalConfig.StationVariant = 6 THEN
	            #sUDT_Handshake_241C := #sUDT_Handshake_141C;
	            #sUDT_Handshake_241D := #sUDT_Handshake_041D;

	        END_IF;


	        #sFB_RightAngledTransfer_241(iUDT_Configuration              := #iqUDT_Configuration."241".RightAngledTransfer,
	                                     iUDT_LowerConveyorConfiguration := #iqUDT_Configuration."240".Conveyor,
	                                     iUDT_UpperConveyorConfiguration := #iqUDT_Configuration."241".Conveyor,
	                                     iUDT_PECConfiguration           := #iqUDT_Configuration."240".PEC_EoS,
	                                     ii_DestinationA                 := #si_240DestinationA,
	                                     ii_DestinationB                 := #si_240DestinationB,
	                                     ii_DestinationC                 := #si_240DestinationC,
	                                     ii_DestinationD                 := #si_240DestinationD,
	                                     ix_HardwareOk                   := #iUDT_HardwareOk."240",
	                                     ix_400vOk                       := #ix_400vOk,
	                                     ix_24vOk                        := #ix_24vOk,
	                                     ix_SafetyOk                     := #ix_SafetyOk,
	                                     ix_AirPressureOk                := #ix_AirPressureOk,
	                                     ix_SectionIsDown                := #ix_SectionIsDown241,
	                                     ix_SectionIsUp                  := #ix_SectionIsUp241,
	                                     ix_ConveyorAAuto                := #iqUDT_WorkstationCommonStatus."230".AutoON,
	                                     ix_ConveyorBAuto                := #iqUDT_WorkstationCommonStatus."250".AutoON,
	                                     ix_ConveyorCAuto                := (#iqUDT_WorkstationCommonStatus."141".AutoON AND (#iqUDT_Configuration.GlobalConfig.StationVariant = 2 OR #iqUDT_Configuration.GlobalConfig.StationVariant = 4 OR #iqUDT_Configuration.GlobalConfig.StationVariant = 6))
	                                     OR (#iqUDT_WorkstationCommonStatus."041".AutoON AND (#iqUDT_Configuration.GlobalConfig.StationVariant = 1 OR #iqUDT_Configuration.GlobalConfig.StationVariant = 3 OR #iqUDT_Configuration.GlobalConfig.StationVariant = 5)),
	                                     ix_ConveyorDAuto                := (#iqUDT_WorkstationCommonStatus."041".AutoON AND (#iqUDT_Configuration.GlobalConfig.StationVariant = 2 OR #iqUDT_Configuration.GlobalConfig.StationVariant = 4 OR #iqUDT_Configuration.GlobalConfig.StationVariant = 6))
	                                     OR (#iqUDT_WorkstationCommonStatus."141".AutoON AND (#iqUDT_Configuration.GlobalConfig.StationVariant = 1 OR #iqUDT_Configuration.GlobalConfig.StationVariant = 3 OR #iqUDT_Configuration.GlobalConfig.StationVariant = 5)),
	                                     ix_PEC                          := #iUDT_MotorInput240.AllSensorPortInputs.LeftSensor,
	                                     ix_ExternalReceiveRequestA      := NOT #iqUDT_WorkstationStatus."230".PEC_EoS.PEC AND #sx_Enable2X0In,
	                                     ix_ExternalReceiveRequestB      := false,
	                                     ix_ExternalReceiveRequestC      := (#sFB_RightAngledTransfer_141.qx_ExternalSendRequestC AND (#iqUDT_Configuration.GlobalConfig.StationVariant = 2 OR #iqUDT_Configuration.GlobalConfig.StationVariant = 4 OR #iqUDT_Configuration.GlobalConfig.StationVariant = 6))
	                                     OR (#sFB_RightAngledTransfer_041.qx_ExternalSendRequestC AND (#iqUDT_Configuration.GlobalConfig.StationVariant = 1 OR #iqUDT_Configuration.GlobalConfig.StationVariant = 3 OR #iqUDT_Configuration.GlobalConfig.StationVariant = 5)),
	                                     ix_ExternalReceiveRequestD      := (#sFB_RightAngledTransfer_041.qx_ExternalSendRequestD AND (#iqUDT_Configuration.GlobalConfig.StationVariant = 2 OR #iqUDT_Configuration.GlobalConfig.StationVariant = 4 OR #iqUDT_Configuration.GlobalConfig.StationVariant = 6))
	                                     OR (#sFB_RightAngledTransfer_141.qx_ExternalSendRequestD AND (#iqUDT_Configuration.GlobalConfig.StationVariant = 1 OR #iqUDT_Configuration.GlobalConfig.StationVariant = 3 OR #iqUDT_Configuration.GlobalConfig.StationVariant = 5)),
	                                     ix_PECInfeedA                   := #iqUDT_WorkstationStatus."230".PEC_EoS.PEC,
	                                     ix_PECInfeedC                   := (#iqUDT_WorkstationStatus."140".PEC_EoS.PEC AND (#iqUDT_Configuration.GlobalConfig.StationVariant = 2 OR #iqUDT_Configuration.GlobalConfig.StationVariant = 4 OR #iqUDT_Configuration.GlobalConfig.StationVariant = 6))
	                                     OR (#iqUDT_WorkstationStatus."040".PEC_EoS.PEC AND (#iqUDT_Configuration.GlobalConfig.StationVariant = 1 OR #iqUDT_Configuration.GlobalConfig.StationVariant = 3 OR #iqUDT_Configuration.GlobalConfig.StationVariant = 5)),
	                                     ix_PECInfeedD                   := (#iqUDT_WorkstationStatus."040".PEC_EoS.PEC AND (#iqUDT_Configuration.GlobalConfig.StationVariant = 2 OR #iqUDT_Configuration.GlobalConfig.StationVariant = 4 OR #iqUDT_Configuration.GlobalConfig.StationVariant = 6))
	                                     OR (#iqUDT_WorkstationStatus."140".PEC_EoS.PEC AND (#iqUDT_Configuration.GlobalConfig.StationVariant = 1 OR #iqUDT_Configuration.GlobalConfig.StationVariant = 3 OR #iqUDT_Configuration.GlobalConfig.StationVariant = 5)),
	                                     qUDT_HMIRATStatus               => #iqUDT_WorkstationStatus."241".RightAngledTransfer,
	                                     qUDT_HMIConveyorStatus          => #iqUDT_WorkstationStatus."240".Conveyor,
	                                     qUDT_HMIPECStatus               => #iqUDT_WorkstationStatus."240".PEC_EoS,
	                                     qUDT_RATStatus                  => #iqUDT_WorkstationCommonStatus."241",
	                                     qUDT_ConveyorStatus             => #iqUDT_WorkstationCommonStatus."240",
	                                     qx_PopupControl                 => #qx_PopupControl241,
	                                     iqUDT_EquipmentControl          := #iqUDT_EquipmentControl,
	                                     iqUDT_RATCommand                := #iqUDT_WorkstationCommands."241".RightAngledTransfer,
	                                     iqUDT_ConveyorCommand           := #iqUDT_WorkstationCommands."240".Conveyor,
	                                     iqUDT_RATStatistics             := #iqUDT_WorkstationStatistics."241".RightAngledTransfer,
	                                     iqUDT_ConveyorStatistics        := #iqUDT_WorkstationStatistics."240".Conveyor,
	                                     iqUDT_PECStatistics             := #iqUDT_WorkstationStatistics."240".PEC_EoS,
	                                     iqUDT_HandShakeConveyorA        := #sUDT_Handshake_230,
	                                     iqUDT_HandShakeConveyorB        := #sUDT_Handshake_240,
	                                     iqUDT_HandShakeConveyorC        := #sUDT_Handshake_241C,
	                                     iqUDT_HandShakeConveyorD        := #sUDT_Handshake_241D,
	                                     iqUDT_LowerConveyorInterface    := #sUDT_Interface_240,
	                                     iqUDT_UpperConveyorInterface    := #sUDT_Interface_241,
	                                     iqUDT_RATPositioning            := #iqUDT_RATPositioning240,
	                                     iqUDT_BladeStopEoSInterface     := #tUDT_DummyBladeStop,
	                                     iqUDT_BladeStopBoSInterface     := #tUDT_DummyBladeStop);

	    END_REGION

	    IF #iqUDT_Configuration.GlobalConfig.StationVariant = 1 OR #iqUDT_Configuration.GlobalConfig.StationVariant = 3 OR #iqUDT_Configuration.GlobalConfig.StationVariant = 5 THEN
	        #sUDT_Handshake_041C := #sUDT_Handshake_241C;
	        #sUDT_Handshake_141D := #sUDT_Handshake_241D;
	    ELSIF #iqUDT_Configuration.GlobalConfig.StationVariant = 2 OR #iqUDT_Configuration.GlobalConfig.StationVariant = 4 OR #iqUDT_Configuration.GlobalConfig.StationVariant = 6 THEN
	        #sUDT_Handshake_141C := #sUDT_Handshake_241C;
	        #sUDT_Handshake_041D := #sUDT_Handshake_241D;

	    END_IF;


	    REGION MCO

	        #sFB_MCOConveyLinxAixController_241(iUDT_AixConfig          := #iqUDT_Configuration."241".MCO_M01,
	                                            iv_AixInputsModule    := #iUDT_MotorInput240,
	                                            ii_PositionSetpoint     := #iqUDT_RATPositioning240.Upper.EndPosition,
	                                            ix_24vOk                := #ix_24vOk,
	                                            ix_SimulationModeActive := "DB_Memory".Simulation,
	                                            ii_MotorPositionId      := 2,
	                                            ix_StartPositioning     := #iqUDT_RATPositioning240.Upper.Start,
	                                            ix_ResetPosition        := #iqUDT_RATPositioning240.Upper.ResetPosition,
	                                            qUDT_HMIStatus          => #iqUDT_WorkstationStatus."241".MCO_M01,
	                                            qx_Positioned           => #iqUDT_RATPositioning240.Upper.Done,
	                                            iqv_AixOutputsModule  := #iqUDT_MotorOutput240,
	                                            iqUDT_ConveyorInterface := #sUDT_Interface_241,
	                                            iqUDT_MCOStatistics     := #iqUDT_WorkstationStatistics."241".MCO_M01);
	    END_REGION

	END_REGION

	REGION 250

	    REGION Displacement
	        #sFB_Displacement250(#sUDT_Interface_250);
	    END_REGION



	    REGION EoS


	        #sFB_PEC_250(ix_PEC                  := #iUDT_MotorInput250.AllSensorPortInputs.LeftSensor,
	                     iUDT_PECConfiguration   := #iqUDT_Configuration."250".PEC_EoS,
	                     qUDT_HMIStatus          => #iqUDT_WorkstationStatus."250".PEC_EoS,
	                     iqUDT_ConveyorInterface := #sUDT_Interface_250,
	                     iqUDT_PECStatistics     := #iqUDT_WorkstationStatistics."250".PEC_EoS);




	    END_REGION

	    REGION Conveyor

	        #sFB_Conveyor_250(iUDT_ConveyorConfiguration := #iqUDT_Configuration."250".Conveyor,
	                          idi_PECEoSDistance         := 0,
	                          idi_PECBoSDistance         := 0,
	                          ii_ExternalSpeed           := 0,
	                          ix_SafetyOk                := #ix_SafetyOk,
	                          ix_24vOk                   := #ix_24vOk,
	                          ix_400vOk                  := #ix_400vOk,
	                          ix_HardwareOk              := #iUDT_HardwareOk."250",
	                          ix_PECEoS                  := #iqUDT_WorkstationStatus."250".PEC_EoS.PEC,
	                          ix_PECBoS                  := TRUE,
	                          ix_ReverseDirection        := FALSE,
	                          ix_ExternalRequestDieBack  := FALSE,
	                          ix_ExternalRequestHold     := FALSE,
	                          ix_ResetEnergySave         := FALSE,
	                          qUDT_HMIStatus             => #iqUDT_WorkstationStatus."250".Conveyor,
	                          qUDT_Status                => #iqUDT_WorkstationCommonStatus."250",
	                          iqUDT_EquipmentControl     := #iqUDT_EquipmentControl,
	                          iqUDT_ConveyorCommand      := #iqUDT_WorkstationCommands."250".Conveyor,
	                          iqUDT_ConveyorInterface    := #sUDT_Interface_250,
	                          iqUDT_HandShakeUp          := #sUDT_Handshake_240,
	                          iqUDT_HandShake            := #sUDT_Handshake_250,
	                          iqUDT_Statistics           := #iqUDT_WorkstationStatistics."250".Conveyor);

	    END_REGION

	    REGION MCO

	        #sFB_MCOConveyLinxAixController_250(iUDT_AixConfig          := #iqUDT_Configuration."250".MCO_M01,
	                                            iv_AixInputsModule    := #iUDT_MotorInput250,
	                                            ix_24vOk                := #ix_24vOk,
	                                            ix_SimulationModeActive := "DB_Memory".Simulation,
	                                            ii_MotorPositionId      := 1,
	                                            qUDT_HMIStatus          => #iqUDT_WorkstationStatus."250".MCO_M01,
	                                            iqv_AixOutputsModule  := #iqUDT_MotorOutput250,
	                                            iqUDT_ConveyorInterface := #sUDT_Interface_250,
	                                            iqUDT_MCOStatistics     := #iqUDT_WorkstationStatistics."250".MCO_M01);
	    END_REGION

	END_REGION

	REGION 260

	    REGION Displacement
	        #sFB_Displacement260(#sUDT_Interface_260);
	    END_REGION

	    REGION Tracking

	        #sFB_Tracking_260(iUDT_ConveyorCommonConfiguration := #iqUDT_Configuration."260".Conveyor.Common,
	                          iqa_TrackingData                 := #sa_TrackingArray_260,
	                          iqUDT_ConveyorInterface          := #sUDT_Interface_260,
	                          iqUDT_HandshakeUp                := #sUDT_Handshake_250,
	                          iqUDT_Handshake                  := #sUDT_Handshake_260);

	    END_REGION

	    REGION EoS

	        #sFB_PECUpdate_260(iUDT_PECUpdateConfiguration      := #iqUDT_Configuration."260".PEC_EoS,
	                           iUDT_ConveyorCommonConfiguration := #iqUDT_Configuration."260".Conveyor.Common,
	                           ix_PEC                           := #iUDT_MotorInput250.AllSensorPortInputs.RightSensor,
	                           ix_TeachingMode                  := FALSE,
	                           qUDT_Status                      => #iqUDT_WorkstationStatus."260".PEC_EoS,
	                           iqUDT_ConveyorInterface          := #sUDT_Interface_260,
	                           iqUDT_UnknownGINRange            := #iqUDT_UnknownGINRange,
	                           iqUDT_FifoHeader                 := #sUDT_FifoLostGINHeader,
	                           iqUDT_Statistics                 := #iqUDT_WorkstationStatistics."260".PEC_EoS,
	                           iqa_TrackingData                 := #sa_TrackingArray_260,
	                           iqa_FifoData                     := #sa_FifoLostGINData);




	    END_REGION

	    REGION Conveyor

	        #sFB_Conveyor_260(iUDT_ConveyorConfiguration := #iqUDT_Configuration."260".Conveyor,
	                          idi_PECEoSDistance         := 0,
	                          idi_PECBoSDistance         := 0,
	                          ii_ExternalSpeed           := 0,
	                          ix_SafetyOk                := #ix_SafetyOk,
	                          ix_24vOk                   := #ix_24vOk,
	                          ix_400vOk                  := #ix_400vOk,
	                          ix_HardwareOk              := #iUDT_HardwareOk."250",
	                          ix_PECEoS                  := #iqUDT_WorkstationStatus."260".PEC_EoS.PEC,
	                          ix_PECBoS                  := TRUE,
	                          ix_ReverseDirection        := FALSE,
	                          ix_ExternalRequestDieBack  := FALSE,
	                          ix_ExternalRequestHold     := FALSE,
	                          ix_ResetEnergySave         := FALSE,
	                          qUDT_HMIStatus             => #iqUDT_WorkstationStatus."260".Conveyor,
	                          qUDT_Status                => #iqUDT_WorkstationCommonStatus."260",
	                          iqUDT_EquipmentControl     := #iqUDT_EquipmentControl,
	                          iqUDT_ConveyorCommand      := #iqUDT_WorkstationCommands."260".Conveyor,
	                          iqUDT_ConveyorInterface    := #sUDT_Interface_260,
	                          iqUDT_HandShakeUp          := #sUDT_Handshake_250,
	                          iqUDT_HandShake            := #sUDT_Handshake_260,
	                          iqUDT_Statistics           := #iqUDT_WorkstationStatistics."260".Conveyor);

	    END_REGION

	    REGION MCO

	        #sFB_MCOConveyLinxAixController_260(iUDT_AixConfig          := #iqUDT_Configuration."260".MCO_M01,
	                                            iv_AixInputsModule    := #iUDT_MotorInput250,
	                                            ix_24vOk                := #ix_24vOk,
	                                            ix_SimulationModeActive := "DB_Memory".Simulation,
	                                            ii_MotorPositionId      := 2,
	                                            qUDT_HMIStatus          => #iqUDT_WorkstationStatus."260".MCO_M01,
	                                            iqv_AixOutputsModule  := #iqUDT_MotorOutput250,
	                                            iqUDT_ConveyorInterface := #sUDT_Interface_260,
	                                            iqUDT_MCOStatistics     := #iqUDT_WorkstationStatistics."260".MCO_M01);
	    END_REGION

	END_REGION

	REGION 270

	    REGION Displacement
	        #sFB_Displacement270(#sUDT_Interface_270);
	    END_REGION

	    REGION Tracking

	        #sFB_Tracking_270(iUDT_ConveyorCommonConfiguration := #iqUDT_Configuration."270".Conveyor.Common,
	                          iqa_TrackingData                 := #sa_TrackingArray_270,
	                          iqUDT_ConveyorInterface          := #sUDT_Interface_270,
	                          iqUDT_HandshakeUp                := #sUDT_Handshake_260,
	                          iqUDT_Handshake                  := #iqUDT_HandshakeDownstream270);

	    END_REGION

	    REGION EoS

	        #sFB_PECUpdate_270(iUDT_PECUpdateConfiguration      := #iqUDT_Configuration."270".PEC_EoS,
	                           iUDT_ConveyorCommonConfiguration := #iqUDT_Configuration."270".Conveyor.Common,
	                           ix_PEC                           := #iUDT_MotorInput270.AllSensorPortInputs.LeftSensor,
	                           ix_TeachingMode                  := FALSE,
	                           qUDT_Status                      => #iqUDT_WorkstationStatus."270".PEC_EoS,
	                           iqUDT_ConveyorInterface          := #sUDT_Interface_270,
	                           iqUDT_UnknownGINRange            := #iqUDT_UnknownGINRange,
	                           iqUDT_FifoHeader                 := #sUDT_FifoLostGINHeader,
	                           iqUDT_Statistics                 := #iqUDT_WorkstationStatistics."270".PEC_EoS,
	                           iqa_TrackingData                 := #sa_TrackingArray_270,
	                           iqa_FifoData                     := #sa_FifoLostGINData);

	    END_REGION

	    REGION Conveyor

	        #iqUDT_HandshakeDownstream270.RTR := #iqUDT_HandshakeDownstream270.RTR OR #iqUDT_WorkstationStatus."270".PEC_EoS.PEC;

	        #sFB_Conveyor_270(iUDT_ConveyorConfiguration := #iqUDT_Configuration."270".Conveyor,
	                          idi_PECEoSDistance         := #iqUDT_Configuration."270".PEC_EoS.Distance,
	                          idi_PECBoSDistance         := 0,
	                          ii_ExternalSpeed           := 0,
	                          ix_SafetyOk                := #ix_SafetyOk,
	                          ix_24vOk                   := #ix_24vOk,
	                          ix_400vOk                  := #ix_400vOk,
	                          ix_HardwareOk              := #iUDT_HardwareOk."270",
	                          ix_PECEoS                  := #iqUDT_WorkstationStatus."270".PEC_EoS.PEC,
	                          ix_PECBoS                  := TRUE,
	                          ix_ReverseDirection        := FALSE,
	                          ix_ExternalRequestDieBack  := FALSE,
	                          ix_ExternalRequestHold     := FALSE,
	                          ix_ResetEnergySave         := FALSE,
	                          qUDT_HMIStatus             => #iqUDT_WorkstationStatus."270".Conveyor,
	                          qUDT_Status                => #iqUDT_WorkstationCommonStatus."270",
	                          iqUDT_EquipmentControl     := #iqUDT_EquipmentControl,
	                          iqUDT_ConveyorCommand      := #iqUDT_WorkstationCommands."270".Conveyor,
	                          iqUDT_ConveyorInterface    := #sUDT_Interface_270,
	                          iqUDT_HandShakeUp          := #sUDT_Handshake_260,
	                          iqUDT_HandShake            := #iqUDT_HandshakeDownstream270,
	                          iqUDT_Statistics           := #iqUDT_WorkstationStatistics."270".Conveyor);

	    END_REGION

	    REGION MCO

	        #sFB_MCOConveyLinxAixController_270(iUDT_AixConfig          := #iqUDT_Configuration."270".MCO_M01,
	                                            iv_AixInputsModule    := #iUDT_MotorInput270,
	                                            ix_24vOk                := #ix_24vOk,
	                                            ix_SimulationModeActive := "DB_Memory".Simulation,
	                                            ii_MotorPositionId      := 1,
	                                            qUDT_HMIStatus          => #iqUDT_WorkstationStatus."270".MCO_M01,
	                                            iqv_AixOutputsModule  := #iqUDT_MotorOutput270,
	                                            iqUDT_ConveyorInterface := #sUDT_Interface_270,
	                                            iqUDT_MCOStatistics     := #iqUDT_WorkstationStatistics."270".MCO_M01);
	    END_REGION

	END_REGION

END_FUNCTION_BLOCK

